PROGRAM VariableHandleForHmi
VAR
END_VAR

numberOfOpenWindows := EnOcean.totalNumberOfWindowsOpen;
boardroomModeIsProjector := LightControl.xBoardToom_Lights_ProjectorMode;
boardroomModeIsFullOn := PTM200StrippedTables[3].Signal OR PTM200StrippedTables[2].Signal;
communalOccupancy1 := Dali.CommunalAreaPIR_1_Occupancy;
communalOccupancy2 := Dali.CommunalAreaPIR_2_Occupancy;
staffOccupancy1 := Dali.StaffroomPIR_1_Occupancy;
staffOccupancy2 := Dali.StaffroomPIR_2_Occupancy;
boardOccupancy1 := Dali.BoardroomPIR_1_Occupancy;
boardOccupancy2 := Dali.BoardroomPIR_2_Occupancy;
communalLux1 := Dali.CommunalAreaPIR_1_LuxLevel;
communalLux2 := Dali.CommunalAreaPIR_2_LuxLevel;
staffLux1 := Dali.StaffroomPIR_1_LuxLevel;
staffLux2 := Dali.StaffroomPIR_2_LuxLevel;
boardLux1 := Dali.BoardroomPIR_1_LuxLevel;
boardLux2 := Dali.BoardroomPIR_2_LuxLevel;

END_PROGRAM

(* stored: Version 1.1.0.1, ProductVersion 3.1.4024.12
   POU VariableHandleForHmi: Id {de9878e5-2b3a-4989-a664-6eb3d99a800d}, SpecialFunc None *)
